Universal Robots URScript: custom_script_1.urscript

# HEADER_BEGIN
DATA_SIZE = 6
global stop_execution = 0
DUMMY_RETURN_VALUE = 199
MULTIPLICATION_SCALING_FACTOR = 1000000

global delta_xz=0.05
global DrillDepthSet={{DRILL_DEPTH_SET_REPLACE}}
global PressForceSet=110
global DrillTimeSet=7.5
global ForceDampingSet=0.07
global Nz=0
global Nx=0
global Loop_active=True

global Pos1= get_actual_tcp_pose ()

thread comm_thread():
  textmsg("Entering Comm Thread")

  while stop_execution == 0:
    enter_critical
    data = socket_read_binary_integer(DATA_SIZE, "sharing_socket")
    if data[0] > 0:
      var1 = data[1]/MULTIPLICATION_SCALING_FACTOR
      DrillDepthSet = var1
      stop_execution = data[6]/MULTIPLICATION_SCALING_FACTOR
      if stop_execution == 1:
        Loop_active=False
      end
    end
    socket_send_int(DUMMY_RETURN_VALUE, "sharing_socket")
    exit_critical
  end
end

thread move_thread():
  Pos1= get_actual_tcp_pose()
  while (Loop_active):
    Pos1[1] = Pos1[1] - DrillDepthSet
    movel(Pos1, a=1.2, v=0.25)
    Pos1[1] = Pos1[1] + DrillDepthSet
    movel(Pos1, a=1.2, v=0.25)
  end
end

def updown():
  main_comm_thread = run comm_thread()
  main_move_thread = run move_thread()
  join main_move_thread
  join main_comm_thread
end


# HEADER_END


set_tcp(p[0.0,0.0,0.212,0.0,0.0,0.0])
set_target_payload(0.500000, [0.000000, 0.000000, 0.020000], [0.000485, 0.000485, 0.000485, 0.000000, 0.000000, 0.000000])
set_safety_mode_transition_hardness(1)
set_gravity([0.0, -9.82, 6.013015783813504E-16])
set_tool_communication(False, 115200, 0, 1, 1.5, 3.5)
set_tool_output_mode(0)
set_tool_digital_output_mode(0, 1)
set_tool_digital_output_mode(1, 1)
set_tool_voltage(0)
set_standard_analog_input_domain(0, 1)
set_standard_analog_input_domain(1, 1)
set_tool_analog_input_domain(0, 1)
set_tool_analog_input_domain(1, 1)
set_analog_outputdomain(0, 0)
set_analog_outputdomain(1, 0)
set_input_actions_to_default()

textmsg("Establishing connection...")
connection_status = socket_open("192.168.56.1", 30003, "sharing_socket")

if connection_status == True:

  textmsg("Connection established successfully.")

  updown()

  textmsg("Exiting main while loop in the custom script")

else:

  textmsg("Could not establish connection.")

end

# join thread_custom

socket_close("sharing_socket")
